FUNCTION_BLOCK Recipe_20014_chocoCookie
VAR_INPUT
	TaskID	: 	LREAL;
	Execute :	BOOL;
END_VAR
VAR_OUTPUT
	Test		: INT;
	RecipeDone	: BOOL;
	InitDone	: BOOL;
	RecipeInfo	: DUT_RECIPEOFFER;
END_VAR
VAR	
	Done		: BOOL;
	
	
	
END_VAR

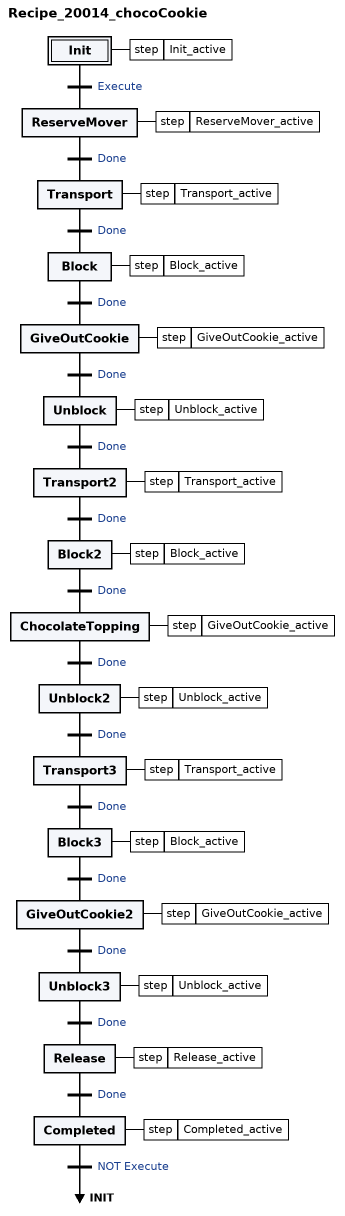
INITIAL_STEP Init:
    Init_active(N);  // step action
END_STEP
TRANSITION FROM Init TO ReserveMover
    := Execute;
END_TRANSITION
STEP ReserveMover:
    ReserveMover_active(N);  // step action
END_STEP
TRANSITION FROM ReserveMover TO Transport
    := Done;
END_TRANSITION
STEP Transport:
    Transport_active(N);  // step action
END_STEP
TRANSITION FROM Transport TO Block
    := Done;
END_TRANSITION
STEP Block:
    Block_active(N);  // step action
END_STEP
TRANSITION FROM Block TO GiveOutCookie
    := Done;
END_TRANSITION
STEP GiveOutCookie:
    GiveOutCookie_active(N);  // step action
END_STEP
TRANSITION FROM GiveOutCookie TO Unblock
    := Done;
END_TRANSITION
STEP Unblock:
    Unblock_active(N);  // step action
END_STEP
TRANSITION FROM Unblock TO Transport2
    := Done;
END_TRANSITION
STEP Transport2:
    Transport_active(N);  // step action
END_STEP
TRANSITION FROM Transport2 TO Block2
    := Done;
END_TRANSITION
STEP Block2:
    Block_active(N);  // step action
END_STEP
TRANSITION FROM Block2 TO ChocolateTopping
    := Done;
END_TRANSITION
STEP ChocolateTopping:
    GiveOutCookie_active(N);  // step action
END_STEP
TRANSITION FROM ChocolateTopping TO Unblock2
    := Done;
END_TRANSITION
STEP Unblock2:
    Unblock_active(N);  // step action
END_STEP
TRANSITION FROM Unblock2 TO Transport3
    := Done;
END_TRANSITION
STEP Transport3:
    Transport_active(N);  // step action
END_STEP
TRANSITION FROM Transport3 TO Block3
    := Done;
END_TRANSITION
STEP Block3:
    Block_active(N);  // step action
END_STEP
TRANSITION FROM Block3 TO GiveOutCookie2
    := Done;
END_TRANSITION
STEP GiveOutCookie2:
    GiveOutCookie_active(N);  // step action
END_STEP
TRANSITION FROM GiveOutCookie2 TO Unblock3
    := Done;
END_TRANSITION
STEP Unblock3:
    Unblock_active(N);  // step action
END_STEP
TRANSITION FROM Unblock3 TO Release
    := Done;
END_TRANSITION
STEP Release:
    Release_active(N);  // step action
END_STEP
TRANSITION FROM Release TO Completed
    := Done;
END_TRANSITION
STEP Completed:
    Completed_active(N);  // step action
END_STEP
TRANSITION FROM Completed TO INIT
    := NOT Execute;
END_TRANSITION

ACTION Release_active:
Done := FALSE;


ExecuteSkill.SkillID 			:= 1311;
ExecuteSkill.SkillName	 		:= 'Release Mover';
ExecuteSkill.Parameter[1].ID 	:= 1;
ExecuteSkill.Parameter[1].Name 	:= 'TaskID';
ExecuteSkill.Parameter[1].Value := TaskID;
ExecuteSkill();

Done := TRUE;
END_ACTION

ACTION Unblock_active:
Done := FALSE;

//Skill auswählen
ExecuteSkill.SkillID := 1316;
ExecuteSkill.SkillName	 := 'Unblock Mover';

//Parameter setzen
ExecuteSkill.Parameter[1].ID := 1;
ExecuteSkill.Parameter[1].Name := 'TaskID';
ExecuteSkill.Parameter[1].Value := TaskID;

//Skill hinzufügen
ExecuteSkill();


Done := TRUE;
END_ACTION

ACTION Transport_active:
Done := FALSE;

//Skill auswählen
ExecuteSkill.SkillID 		:= 1320;
ExecuteSkill.SkillName	 	:= 'Transport Mover';

//Geschwindigkeit setzen
ExecuteSkill.Parameter[1].ID := 3;
ExecuteSkill.Parameter[1].Name := 'Velocity';
ExecuteSkill.Parameter[1].Value := 3000;


ExecuteSkill();

Done := ExecuteSkill.Done;
END_ACTION

ACTION Done_active:
Done := TRUE;
END_ACTION

ACTION Init_active:
RecipeDone := FALSE;

// Initialisation of Recipe Parameters an name etc
RecipeInfo.Name := 'Simple Chocolate Cookie';
RecipeInfo.Description := 'This Recipe produces a simple, but still delicious two-layer Cookie with Chocolate inside';
RecipeInfo.Dummy := FALSE;
RecipeInfo.RecipeID := 10014;

Initdone := TRUE;


//Parameter 1:
(*
	RecipeInfo.UserParameter[1].Dummy 		:= 
	RecipeInfo.UserParameter[1].Default		:=
	RecipeInfo.UserParameter[1].Description	:=
	RecipeInfo.UserParameter[1].MaxValue	:=
	RecipeInfo.UserParameter[1].MinValue	:=
	RecipeInfo.UserParameter[1].Name		:=
	RecipeInfo.UserParameter[1].Unit		:=
*)
//Parameter 2:

(*
	RecipeInfo.UserParameter[2].Dummy 		:= 
	RecipeInfo.UserParameter[2].Default		:=
	RecipeInfo.UserParameter[2].Description	:=
	RecipeInfo.UserParameter[2].MaxValue	:=
	RecipeInfo.UserParameter[2].MinValue	:=
	RecipeInfo.UserParameter[2].Name		:=
	RecipeInfo.UserParameter[2].Unit		:=
*)

//Parameter 3:

(*
	RecipeInfo.UserParameter[3].Dummy 		:= 
	RecipeInfo.UserParameter[3].Default		:=
	RecipeInfo.UserParameter[3].Description	:=
	RecipeInfo.UserParameter[3].MaxValue	:=
	RecipeInfo.UserParameter[3].MinValue	:=
	RecipeInfo.UserParameter[3].Name		:=
	RecipeInfo.UserParameter[3].Unit		:=
*)

//Parameter 4:

(*
	RecipeInfo.UserParameter[4].Dummy 		:= 
	RecipeInfo.UserParameter[4].Default		:=
	RecipeInfo.UserParameter[4].Description	:=
	RecipeInfo.UserParameter[4].MaxValue	:=
	RecipeInfo.UserParameter[4].MinValue	:=
	RecipeInfo.UserParameter[4].Name		:=
	RecipeInfo.UserParameter[4].Unit		:=
*)


//Parameter 5:

(*
	RecipeInfo.UserParameter[5].Dummy 		:= 
	RecipeInfo.UserParameter[5].Default		:=
	RecipeInfo.UserParameter[5].Description	:=
	RecipeInfo.UserParameter[5].MaxValue	:=
	RecipeInfo.UserParameter[5].MinValue	:=
	RecipeInfo.UserParameter[5].Name		:=
	RecipeInfo.UserParameter[5].Unit		:=
*)
END_ACTION

ACTION Completed_active:
RecipeDone := TRUE;
Done := FALSE;
END_ACTION

ACTION GiveOutCookie_active:
Done := FALSE;

ExecuteSkill.SkillID 			:= 1210;
ExecuteSkill.SkillName	 		:= 'Dispense Chocolate Topping';
ExecuteSkill.Parameter[1].ID 	:= 1;
ExecuteSkill.Parameter[1].Name 	:= 'Amount';
ExecuteSkill.Parameter[1].Value := 5.31;
ExecuteSkill();
Done := TRUE;
END_ACTION

ACTION Block_active:
Done := FALSE;

//Skill auswählen
ExecuteSkill.SkillID := 1315;
ExecuteSkill.SkillName	 := 'Block Mover';

//Parameter setzen
ExecuteSkill.Parameter[1].ID := 1;
ExecuteSkill.Parameter[1].Name := 'TaskID';
ExecuteSkill.Parameter[1].Value := TaskID;

//Skill hinzufügen
ExecuteSkill();


Done := TRUE;
END_ACTION

ACTION ReserveMover_active:
Done := FALSE;


ExecuteSkill.SkillID := 1310;
ExecuteSkill.SkillName	 := 'Reserve Mover';
ExecuteSkill.Parameter[1].ID := 1;
ExecuteSkill.Parameter[1].Name := 'TaskID';
ExecuteSkill.Parameter[1].Value := TaskID;
ExecuteSkill();

Done := TRUE;
END_ACTION

END_FUNCTION_BLOCK

(* stored: Version 1.1.0.1, ProductVersion 3.1.0.25
   POU Recipe_20014_chocoCookie: Id {0eb1340f-cf89-42b5-b0c7-f40ef0e8a436}
   Action Release_active: Id {2398d7ba-ec08-43f1-8497-5e68f00ccd29}
   Action Unblock_active: Id {49c2da97-6de4-4ace-aee1-4d500de9b83d}
   Action Transport_active: Id {73fd6147-de43-44e9-8be2-65f118dacf60}
   Action Done_active: Id {8dfcb5a0-5352-44ef-b476-1b6b235b3f79}
   Action Init_active: Id {9d71b8e7-499e-4649-9457-342f2001bca3}
   Action Completed_active: Id {bc9d8d1d-4b44-46ca-8bd2-32853f79f852}
   Action GiveOutCookie_active: Id {d3e6b6f8-d7e1-46f3-9a54-196914eac4bc}
   Action Block_active: Id {e7dc6b0a-b509-4819-a848-f12448e258f0}
   Action ReserveMover_active: Id {efa29c38-401c-48ed-bfd9-a6c9597f2906} *)
